{attribute addProperty BoxType "EP9128-0021-0016"}
{attribute addProperty Id "A_0007_EP9128_0021_0017A_0007_EP9128_0021_0017_447D04D54696587A_0004_EP9128_0021_0016_2_EP9128_1021EP9128_179A0949162"}
{attribute addProperty CRC "1377990989"}
{attribute addProperty SizeInBites "4712"}
{attribute addProperty SizeInBytes "589"}
TYPE A_0004_EP9128_0021_0016_5222794D EXTENDS EP9128_179A0949 :
STRUCT
	{attribute addProperty Name "A_0007_EP9128_0021_0017"}
	A_0007_EP9128_0021_0017 : A_0007_EP9128_0021_0017_447D04D5;
	{attribute addProperty Name "A_0004_EP9128_0021_0016_2_EP9128_1021"}
	A_0004_EP9128_0021_0016_2_EP9128_1021 : EP9128_179A0949;
END_STRUCT
END_TYPE

(* stored: Version 1.2.0.0, ProductVersion 3.1.4024.9
   DUT A_0004_EP9128_0021_0016_5222794D: Id {2f596562-4b16-42f3-8a8b-bf64fef10a3e} *)
